Fanuc KAREL source: ka00065.KL

-- PROVISIONAL review KL for V770-1; original PC SHA256 3607c3169b3385e4feb7b82aa147debfd0ebd002a7d9981131ea4af5b46de3f6
-- Incomplete behavior may be omitted. Consult companion uncertainty JSON. Do not deploy.
PROGRAM KA00065
%NOLOCKGROUP
-- UNRESOLVED_DECL SRC type=000102
-- UNRESOLVED_DECL DST type=000101
BEGIN
  -- UNRESOLVED_PC offsets 5-20; opcodes 2E,22,32,35
  -- UNRESOLVED_PC offsets 25-45; opcodes 49,7E,4A
  -- UNRESOLVED_PC offsets 50-54; opcodes 7F
END KA00065
